(* PLC project abak_app511_10v 0.0.5.project, Abak.IDE Abak.IDE V1.0.0.0 *)
(* stored: creationDateTime 2026-06-29T13:49:17.1967316, modificationDateTime 2026-06-29T10:17:52.4593439 *)

{attribute 'pack_mode' := '1'}
TYPE Coils :
STRUCT
// --- Режимы работы (команды из HMI) ---
xManualMode_Diazo   : BOOL;        // 1. Ручной режим Diazo
xManualMode_Soda    : BOOL;        // 2. Ручной режим Soda
xManualMode_Steam   : BOOL;        // 3. Ручной режим Steam
// --- Управление водой имитатором ---
xWaterValve_AutoMode : BOOL;       // 4. TRUE=Автоматический режим, FALSE=Ручной
xWaterValve_HmiOpen  : BOOL;       // 5. Открытие по кнопке из HMI (в ручном режиме)
xWaterValve_AutoReq  : BOOL;       // 6. Запрос на открытие от автоматики
// --- Сигналы запуска ---
xWaterStart          : BOOL;       // 7. Запуск дозы воды из HMI
xStartHeating_511    : BOOL;       // 8. Запуск прогрева
// --- Сигналы и статусы стадии промывки (Cascade Drain) ---
xStartCoupling_511   : BOOL;       // 9. Запуск с HMI: признак запуска стадии промывки
xCouplingActive_511  : BOOL;       // 10. Статус для HMI: признак "работа идет"
xCouplingDone_511    : BOOL;       // 11. Статус для HMI: признак "успешно готово"
// --- Режим удержания температуры ---
xKeepTempHeating_511 : BOOL;       // 12. TRUE = удержание температуры после нагрева, FALSE = разовый нагрев
// --- Служебные ---
PLC_READ             : BOOL := TRUE; // 13. Флаг чтения PLC
END_STRUCT
END_TYPE

{attribute 'pack_mode' := '4'}
TYPE HoldingRegs : 
STRUCT
// =============================================================
// Модули M7–M9 (MDS AO-2UI) - Управление клапанами (Выходы 4-20мА)
// =============================================================

// --- Управление запорно-регулирующими клапанами (задание 0..100%) ---
AO1_CmdValveDiazo   : REAL;    // 101. Управление клапаном диазосоединения
AO2_CmdValveSoda    : REAL;    // 103. Управление клапаном едкого натра 14%
AO3_CmdValveSteam   : REAL;    // 105. Управление клапаном пара 6 ати

// --- Уставки с панели (ручной режим) ---
rValveManSet_Diazo  : REAL := 0.0;    // 107. Уставка с панели: Диазо
rValveManSet_Soda   : REAL := 0.0;    // 109. Уставка с панели: Сода
rValveManSet_Steam  : REAL := 0.0;    // 111. Уставка с панели: Пар

// --- Переменные для автоматического управления (выходы ПИД-регуляторов) ---
rAutoSet_Diazo      : REAL;           // 113. Выход ПИД расхода диазо
rAutoSet_Soda       : REAL;           // 115. Выход ПИД расхода соды
rAutoSet_Steam      : REAL;           // 117. Выход ПИД расхода пара

// --- Технологические уставки ---
rWaterDose          : REAL := 5.0;    // 119. Заданная доза воды, м³ (5 кубов)
rSetTempApp511      : REAL := 86.0;   // 121. Уставка температуры
rSetFlowDiazo_511   : REAL;           // 123. Уставка мгновенного расхода диазосоединения (до 19 м³/ч)
rSetPh_511          : REAL;           // 125. Целевая уставка pH (9.5..12 ед.)

// --- Настройки алгоритма опустошения емкости (для наладчика) ---
rZeroFlowThreshold_511 : REAL := 0.2; // 127. Порог падения расхода диазо (м³/ч), ниже которого считаем, что емкость пуста
uiEmptyDelaySec_511    : UINT := 20;  // 129. Задержка фиксации пустого трубопровода (сек)

// --- Настройки ПИД-регуляторов (для наладки контуров с HMI) ---
rKp_Diazo_511        : REAL := 1.0;   // 131. Пропорциональный коэффициент контура расхода диазосоединения
rTn_Diazo_511        : REAL := 5.0;   // 133. Время интегрирования контура расхода диазосоединения (сек)
rKp_pH_511           : REAL := 2.0;   // 135. Пропорциональный коэффициент контура pH
rTn_pH_511           : REAL := 10.0;  // 137. Время интегрирования контура pH (сек)
rKp_Steam_511        : REAL := 2.0;   // 139. Пропорциональный коэффициент контура пара (нагрева)
rTn_Steam_511        : REAL := 15.0;  // 141. Время интегрирования контура пара (сек)
rTv_Steam_511        : REAL := 0.0;   // 143. Время дифференцирования контура пара (сек)

END_STRUCT
END_TYPE

{attribute 'pack_mode' := '4'}
TYPE InputRegs : 
STRUCT
	COILS : DINT := 0;
	INPUTS: DINT := 0;
	HOLDINGS: DINT := 0;
	INPUTREGS: DINT := 0;
	
  // МОДУЛЬ АНАЛОГОВЫХ ВХОДОВ (AI)
  	{region M1_K3_AI_10_08_00 }
    // =========================================================================
    // Первые 3 канала: Сигнализация положений (% открытия) клапанов [1, 2]
    (* adr 9 *)  rPosValveDiazo  : REAL; // Канал 1: Обратная связь клапана диазосоединения
    (* adr 11 *) rPosValveSoda   : REAL; // Канал 2: Обратная связь клапана едкого натра 14%
    (* adr 13 *) rPosValveSteam  : REAL; // Канал 3: Обратная связь клапана пара
    
    // Канал 4: рН-метр
    (* adr 15 *) rPhApp511       : REAL; // Канал 4: Показания pH-метра аппарата 511 (диапазон 9,5..12 ед.)
			{endregion}
				 
				 
				 
	{region M5_MDS_3RTD_1 }
	(* adr 17 *) rTempApp511     : REAL; // Температура в аппарате 511 (до 100 С°)
				
   	{endregion}
		 
	{region tenzo tv006c }
	(* adr 19 *) WE_1            : REAL;
	(* adr 21 *) WE_2            : REAL;
		 
   	{endregion}
		 		 
	{region tenzo ELMER }

	(* adr 23 *) IR_FlowSoda   : REAL; // Текущий расход щелочи , л/мин (или м3/ч)
	(* adr 25 *) IR_TotalSoda   : REAL; // Накопленный объем щелочи, л (или м3)
	(* adr 27 *) IR_FlowWater     : REAL; // Текущий расход воды, л/мин (или м3/ч)
	(* adr 29 *) IR_TotalWater   : REAL; // Накопленный объем воды, л (или м3)
		 
    // Выходные сигналы загрузки воды
	(* adr  31*)   rWaterLoaded   : REAL;    // Сколько воды загружено, м³
	(* adr 32*)    rWaterStatus   : REAL;    // Статус загрузки воды: 0=IDLE 1=RUNNING 2=DONE 3=ABORTED
		 
	(* adr  33*)  IR_FlowDiazo   : REAL; // Текущий мгновенный расход диазосоединения (м3/ч) [3]
	(* adr  35*)  IR_TotalDiazo   : REAL; // Текущий расход диазосоединения, л/мин (или м3/ч)
		 
	(* adr  37*)  rDizoStatus   : REAL; // Текущий расход диазосоединения, л/мин (или м3/ч)

	(* adr  39*) rDiazoLoaded   : REAL; // Текущий расход диазосоединения, л/мин (или м3/ч)
rTimeLeft_511:REAL ;///Оставшиеся секунды при падении расхода
	 rStateCode_511:REAL;//
		  
   	{endregion}
		 
END_STRUCT
END_TYPE

{attribute 'pack_mode' := '1'}
TYPE Inputs : 
STRUCT	
			// =============================================================
			// Модуль M11 (MDS DIO-16BD) - Статусы насосов (Дискретные входы)
			// =============================================================
			{region M11 - MDS DIO-16BD (Статусы насосов)}

		
				     
    // Выходная переменная на физическое реле/соленоид
    xWaterValve_Out     : BOOL;  // 1 канал ФЕ
	xWaterValve_SQH :BOOL;
	xWaterValve_SQL   :BOOL;
			{endregion}
END_STRUCT
END_TYPE

TYPE E_InfluxType :
(
    REAL_TYPE,
    INT_TYPE,
    BOOL_TYPE
);
END_TYPE

TYPE E_AO_State :
(
    INIT    := 0,       // Проверка готовности указателей
    IDLE    := 1,       // Ожидание и циклическое обновление
    ERROR   := 99       // Ошибка адресации или данных
) INT;
END_TYPE

{attribute 'qualified_only'}
{attribute 'strict'}
TYPE E_ValveMode :
(
    INIT := 0,
    AUTO := 1,
    MANUAL := 2,
    ERROR := 99
) INT; // Указываем базовый тип для совместимости
END_TYPE

TYPE E_PumpState :
(
    INIT,           // Инициализация и проверка ресурсов
    IDLE,           // Ожидание команды
    START_PULSE,    // Формирование импульса на ПУСК
    STOP_PULSE,     // Формирование импульса на СТОП
    BLIND_WINDOW,   // Окно игнорирования изменений (x2 времени импульса)
    ERROR           // Состояние критической ошибки
);
END_TYPE

TYPE E_TempSourceSelect_for_cube :
(
   AI_T2_Temp_Cube := 0,  // Температура в кубе
    AI_T3_Temp_Packing := 1,  // T3: Температура в нижней части насадки
    AI_T4_Temp_BotCol := 2   // [Канал 1] T4: Температура низа колонны
) INT;
END_TYPE

{attribute 'qualified_only'}
{attribute 'strict'}
TYPE E_ValveState :
(
    INIT    := 0,   // Инициализация указателей
    IDLE    := 1,   // Ожидание выбора режима
    AUTO    := 2,   // Автоматическое управление
    MANUAL  := 3,   // Ручное управление (HMI)
    FAULT   := 99   // Состояние ошибки (например, Null Pointer)
);
END_TYPE

TYPE E_InfluxType_1 :
(
    REAL_TYPE,
    INT_TYPE,
    BOOL_TYPE
);
END_TYPE

// шаг состояния клиента
{attribute 'strict'}
TYPE CLIENT_STATE :
(
	CREATE	:=	 0,
	WAITING	:=	10,
	SEND	:=	20,
	RECEIVE :=  30
);
END_TYPE

TYPE E_REM_State :
(
    INIT,              (* Начальная инициализация и сброс регистров при запуске *)
    OPERATING,         (* Нормальный циклический режим обработки физических данных *)
    RESET_LOGIC,       (* Шаг удержания команды сброса сумматора *)
    ERROR_COMM         (* Состояние аварии связи при отказе Modbus-канала *)
)  := INIT;            (* По умолчанию автомат всегда стартует с шага INIT *)
END_TYPE

TYPE U_WordToReal : UNION
  dwValue : DWORD;  (* Используется для битовых операций *)
  rValue : REAL;  (* Используется для получения результата *)
END_UNION;
END_TYPE

PROGRAM PLC_PRG // Antigravity Sync Test
VAR
    fbElemerREM         : fbElemerREM;
    
    (* Переменные из вкладки Modbus Generic Serial Slave I/O Mapping *)
    Hmi_Flow_Regs    AT %IW67  : ARRAY[0..1] OF WORD; (* Канал 0 (Мгновенный расход) *)
    Hmi_Volume_Regs  AT %IW63  : ARRAY[0..3] OF WORD; (* Канал 1 (Накопленный объем) *)
    xModbusCommError    : BOOL;                 (* Системный флаг ошибки связи с прибором *)
    xHmiResetCmd        : BOOL;                 (* Сигнал сброса сумматора с HMI-панели *)
    
    (* Выходные очищенные технологические переменные *)
    rCurrentFlowRate    : REAL;                 (* Мгновенный расход в систему, куб.м/ч *)
    lrAccumulatedVol    : LREAL;                (* Точный накопленный объем, куб.м *)
    sOperatorMessage    : STRING(255);          (* Сообщение для текстовой строки на панели *)

    fbWater             : FB_WaterLoading;      (* Наш исправленный ФБ дозирования *)
    
    // ============================================================
    // ПЕРЕМЕННЫЕ ДЛЯ ТЕСТИРОВАНИЯ И СИМУЛЯЦИИ СУММАТОРА
    // ============================================================
    xSimEnable          : BOOL := FALSE;        (* Включить режим симуляции (True = подмена датчиков) *)
    rSimFlowSpeed       : REAL := 20.0;         (* Скорость потока при открытом клапане, куб.м/ч *)
    rSimTotalStorage    : REAL := 125.45;       (* Внутренний виртуальный накопительный счетчик куб.м *)
    
    fbSimClock          : TON;                  (* Генератор тактов времени для подсчета объема *)
    rDeltaVolume        : REAL;                 (* Математический шаг приращения за 1 такт *)
    // ============================================================
END_VAR

                  // ================================================================
// 1. ЧТЕНИЕ РЕАЛЬНЫХ ДАННЫХ ИЗ ПОЛЕВЫХ ПРИБОРОВ
// ================================================================
gvl.gInputRegs.IR_TotalSoda := F_ElemerREM_Volume(pBuf := ADR(%IW65));
gvl.gInputRegs.IR_FlowSoda  := F_ElemerREM_Flow(pBuf := ADR(%IW69));
gvl.gInputRegs.rTempApp511  := F_GetReal_BADC(pBuf := ADR(%IW57));


// ================================================================
// 2. ДИНАМИЧЕСКИЙ СИМУЛЯТОР РАСХОДОМЕРА ВОДЫ
// ================================================================
// Тактовый генератор: срабатывает каждые 100 мс (0.1 секунды) для плавности хода счета
fbSimClock(IN := xSimEnable AND NOT fbSimClock.Q, PT := T#100ms);

IF xSimEnable THEN
    // ЕСЛИ СИМУЛЯЦИЯ ВКЛЮЧЕНА:
    
    // Имитируем поведение потока в зависимости от команды на клапан
    IF gvl.gCoils.xWaterValve_AutoReq THEN
        // Клапан открыт автоматикой -> задаем симуляционный расход
        gvl.gInputRegs.IR_FlowWater := rSimFlowSpeed; 
        
        // Расчет приращения сумматора за 100мс: (куб.м/ч * 0.1с) / 3600с
        IF fbSimClock.Q THEN
            rDeltaVolume := (rSimFlowSpeed * 0.1) / 3600.0;
            rSimTotalStorage := rSimTotalStorage + rDeltaVolume;
        END_IF;
    ELSE
        // Клапан закрыт -> поток прекращается
        gvl.gInputRegs.IR_FlowWater := 0.0;
    END_IF;

    // ПОДМЕНЯЕМ значение сумматора результатом симуляции для ФБ дозирования
    gvl.gInputRegs.IR_TotalWater := rSimTotalStorage;

ELSE
    // ЕСЛИ СИМУЛЯЦИЯ ВЫКЛЮЧЕНА (РАБОЧИЙ РЕЖИМ):
    
    // Читаем физический прибор с адреса %IW71 и %IW75
    gvl.gInputRegs.IR_TotalWater := F_ElemerREM_Volume(pBuf := ADR(%IW71));
    gvl.gInputRegs.IR_FlowWater  := F_ElemerREM_Flow(pBuf := ADR(%IW75));
    
    // Мягко синхронизируем симулятор, чтобы при включении тумблера счет не прыгал назад/вперед
    rSimTotalStorage := gvl.gInputRegs.IR_TotalWater;
END_IF;


// ================================================================
// 3. ВЫЗОВ И ПРОВЕРКА ФУНКЦИОНАЛЬНОГО БЛОКА ЗАГРУЗКИ ВОДЫ
// ================================================================
fbWater(
    rTotalVolume := gvl.gInputRegs.IR_TotalWater,        // Сюда идет либо физический объем, либо симуляция
    rDose        := gvl.gHoldingRegs.rWaterDose,         // Заданная уставка дозы (куб.м)
    rDeadband    := 0.05,                                // Упреждение закрытия (0.05 куб.м)
    xStart       := gvl.gCoils.xWaterStart,              // Команда Старт/Стоп
    xMode        := gvl.gCoils.xWaterValve_AutoMode,     // Флаг режима АВТО клапана
    xAutoControl := gvl.gCoils.xWaterValve_AutoReq       // Управление клапаном (выход на открытие)
);

    gvl.gInputRegs.rWaterLoaded:=fbWater.rLoaded;
    gvl.gInputRegs.rWaterStatus:=fbWater.rStatus;
                
END_PROGRAM

FUNCTION AIToFloat : REAL
VAR_INPUT
	In:UINT;
	Lo,Hi:REAL;
END_VAR
VAR
END_VAR

                  AIToFloat:=(UINT_TO_REAL(In)-10000.0)/40000.0*Hi+Lo;
//AIToFloat:=(UINT_TO_REAL(In)-0.0)/50000.0*Hi+Lo;
                
END_FUNCTION

PROGRAM ASK_prg
VAR
Exatract:	FB_ModbusToFloatArray;
pt : POINTER TO  ARRAY [0..5] OF WORD  ;

//M1_K3_AI_10_08_00 AT %IW58: ARRAY [0..7] OF WORD ; 

buff_abak: ARRAY [0..219] OF WORD ; 
buff_MDS: ARRAY [0..219] OF WORD ; 
buffR_1: ARRAY [0..119] OF REAL ; 
start_ad_mds3rtd:INT:=0;
swap_mds3rtd:INT:=6;
start_ad_mds_8UId:INT:=18;
swap_mds_8UI:INT:=16;

AI: FB_AI;


  
	Info : __SYSTEM.VAR_INFO;

    pAddress : POINTER TO BYTE;
	adress:UDINT;
END_VAR

                  //берем  с модуля  M1_K3_AI_10_08_00 значения  и  копируем в промежуточный буфер   
SysMemCpy(ADR(buff_abak), ADR( %IW0), 8 * SIZEOF(WORD));

//берем  с модуля  MDS_3RTD_1  значения  и  копируем в промежуточный буфер   
SysMemCpy(ADR(buff_MDS), ADR( %IW57), 6 * SIZEOF(WORD));


//берем  с  терминала  tv 006
SysMemCpy(ADR(buff_MDS[swap_mds3rtd]), ADR( %IW53), 2* SIZEOF(WORD));

//берем  с  терминала  tv 006
SysMemCpy(ADR(buff_MDS[swap_mds3rtd+2]), ADR( %IW55), 2* SIZEOF(WORD));

Exatract(aDataIn:=buff_MDS,aDataOut=>buffR_1,IQty:=65,iMode:=1);


// 3. Маппинг (Присвоение значений переменным структуры)
// -------------------------------------------------------------

// === Модуль M1 () ===
GVL.gInputRegs. rPosValveDiazo  := AIToFloat(buff_abak[0],0,100); // 
GVL.gInputRegs.rPosValveSoda  := AIToFloat(buff_abak[1],0,100); // 
GVL.gInputRegs.rPosValveSteam  := AIToFloat(buff_abak[2],0,100); // 
GVL.gInputRegs.rPhApp511  := AIToFloat(buff_abak[4],0,14); // 


// === Модуль M5 () ===

GVL.gInputRegs.rTempApp511  :=buffR_1[0];// TT 511
//GVL.gInputRegs.rTempApp511  :=FC_ModbusToRealSwapped(wWord1 := buff_MDS[0], wWord2 := buff_MDS[1]);
// === Модуль M2 () ===
GVL.rCmdValveDiazo := FloatToAI(gvl.gHoldingRegs.AO1_CmdValveDiazo);

GVL.rCmdValveSoda := FloatToAI(gvl.gHoldingRegs.AO2_CmdValveSoda);

GVL.rCmdValveSteam := FloatToAI(gvl.gHoldingRegs.AO3_CmdValveSteam);


// === Модуль M5 (Индексы 0..2) ===
//GVL.gInputRegs.rTempApp511   := buffR_1[0]; // TT 511


//// === весы  tenzo  M1 ===

	//AI(F_WORD_IN:= gvl.WE_1_f, S_WORD_IN:= gvl.WE_1_s, RANGE_CONV:=FALSE, VAL_OUT=> GVL.gInputRegs.WE_1);
GVL.gInputRegs.WE_1:=buffR_1[3];
GVL.gInputRegs.WE_2:=buffR_1[4];
//// === весы  tenzo  M2 ===
//AI(F_WORD_IN:= gvl.WE_2_f, S_WORD_IN:= gvl.WE_2_s, RANGE_CONV:=TRUE, VAL_OUT=> GVL.gInputRegs.WE_2);
                
END_PROGRAM

FUNCTION_BLOCK FB_ModbusToFloatArray
VAR_INPUT
    aDataIn : ARRAY [0..219] OF WORD; // Входной массив (до 120 регистров)
    iQty    : INT := 1;               // Количество FLOAT переменных для обработки (макс 60)
    iMode   : INT := 1;               // Режим: 0=1234, 1=3412 (частый), 2=2143, 3=4321
END_VAR
VAR_OUTPUT
    aDataOut : ARRAY [0..119] OF REAL; // Выходной массив
    xError   : BOOL;                  // Флаг ошибки (если iQty > 60)
END_VAR
VAR
    i : INT;
    uConverter : U_WordToReal;
    wLow : WORD;
    wHigh : WORD;
    wTemp1 : WORD;
    wTemp2 : WORD;
END_VAR

                  
// Сброс ошибки
xError := FALSE;

// Защита от выхода за пределы массива
IF iQty < 1 OR iQty > 120 THEN
    xError := TRUE;
    RETURN;
END_IF

// Основной цикл
FOR i := 0 TO (iQty - 1) DO
    
    // Получаем пару регистров из массива
    // i*2 - это начало пары (0, 2, 4...)
    wTemp1 := aDataIn[i * 2];     // Первый регистр пары
    wTemp2 := aDataIn[(i * 2) + 1]; // Второй регистр пары

    CASE iMode OF
        // ---------------------------------------------------------
        // Mode 0: 1234 (Big Endian) 
        // Порядок: [HighWord] [LowWord]
        // ---------------------------------------------------------
        0: 
            wHigh := wTemp1;
            wLow  := wTemp2;
            
        // ---------------------------------------------------------
        // Mode 1: 3412 (Middle Little / Word Swap) -> САМЫЙ ЧАСТЫЙ для Modbus
        // Порядок: [LowWord] [HighWord]
        // Регистры меняются местами, байты внутри - нет.
        // ---------------------------------------------------------
        1: 
            wHigh := wTemp2;
            wLow  := wTemp1;

        // ---------------------------------------------------------
        // Mode 2: 2143 (Middle Big / Byte Swap)
        // Порядок: [HighWord swapped] [LowWord swapped]
        // Байты меняются местами внутри каждого слова.
        // ---------------------------------------------------------
        2:
            wHigh := ROL(wTemp1, 8); // Меняем байты местами
            wLow  := ROL(wTemp2, 8);
            
        // ---------------------------------------------------------
        // Mode 3: 4321 (Little Endian)
        // Порядок: [LowWord swapped] [HighWord swapped]
        // Полный разворот: меняются и слова, и байты.
        // ---------------------------------------------------------
        3:
            wHigh := ROL(wTemp2, 8);
            wLow  := ROL(wTemp1, 8);
            
        ELSE
            // По умолчанию используем 3412 (как самый популярный)
            wHigh := wTemp2;
            wLow  := wTemp1;
    END_CASE

    // Сборка DWORD из двух слов
    // Сдвигаем старшее слово на 16 бит влево и добавляем младшее
    uConverter.dwValue := SHL(WORD_TO_DWORD(wHigh), 16) OR WORD_TO_DWORD(wLow);
    
    // Запись результата в выходной массив
    aDataOut[i] := uConverter.rValue;
    
END_FOR
                
END_FUNCTION_BLOCK

FUNCTION_BLOCK Check_Block
VAR_INPUT
	State_Mixer : BOOL;
	Weight : REAL;
END_VAR
VAR_OUTPUT
	State_Block : BOOL;
	State_Block_P102 : BOOL; 
END_VAR
VAR
END_VAR

                  IF NOT State_Mixer THEN
	State_Block := TRUE;
ELSE
	State_Block := FALSE;
END_IF;
IF Weight > 3000 THEN
	State_Block_P102 := TRUE;
ELSE 
	State_Block_P102 := FALSE;
END_IF;
                
END_FUNCTION_BLOCK

FUNCTION FloatToAI : UINT
VAR_INPUT
	In:REAL;
	
END_VAR
VAR
END_VAR

                  FloatToAI:=REAL_TO_UINT(In/100.0*40000.0+10000.0);
                
END_FUNCTION

(*
* @fb: PRG_ModbusSlave_Sync
* @desc: Исправленная синхронизация через прямые указатели (устранение C0047/C0077)
*)
PROGRAM PRG_ModbusSlave_Sync
VAR
    fbSlv               : abakplcutils.MDB;
    sStatus             : STRING(255);
    
    // Вспомогательные буферы
    wMbHolding          : ARRAY[0..500] OF WORD; 
    wOldMbHolding       : ARRAY[0..500] OF WORD; 
    
    // Указатели для работы со структурами GVL как с массивами
    pCurrWord           : POINTER TO WORD;
    pOldWord            : POINTER TO WORD;
    
    wIndex              : WORD;
    uiHoldRegsCnt       : WORD;
    uiInRegsCnt         : WORD;
    xFirstLoop          : BOOL := TRUE;
	
    C_INPUT_REG_START   : WORD := 1;
    C_HOLD_REG_START    : WORD := 1000;
END_VAR

                  // 1. Инициализация и расчет длин (через SIZEOF, чтобы не зависеть от типов)
IF xFirstLoop THEN
    uiInRegsCnt   := ANY_TO_WORD(SIZEOF(GVL.gInputRegs) / 2);
    uiHoldRegsCnt := ANY_TO_WORD(SIZEOF(GVL.gHoldingRegs) / 2);
    
    // Предзаполнение Modbus и локального зеркала (используем SysMem для скорости)
    fbSlv.SetWordRegs(reg := C_HOLD_REG_START, pBuf := ADR(GVL.gHoldingRegs), cnt := uiHoldRegsCnt);
    SysMem.SysMemCpy(pDest := ADR(wOldMbHolding), pSrc := ADR(GVL.gHoldingRegs), udiCount := uiHoldRegsCnt * 2);
    
    xFirstLoop := FALSE;
    RETURN;
END_IF

// --- ШАГ 1: Input Registers (Запись всей структуры целиком через указатель) ---
sStatus := 'Обновление Input Registers';
fbSlv.SetWordRegs(reg := C_INPUT_REG_START, pBuf := ADR(GVL.gInputRegs), cnt := uiInRegsCnt);

// --- ШАГ 2: Holding Registers (Синхронизация через пошаговый доступ к памяти) ---
sStatus := 'Синхронизация Holding...';
fbSlv.GetWordRegs(reg := C_HOLD_REG_START, pBuf := ADR(wMbHolding), cnt := uiHoldRegsCnt);

FOR wIndex := 0 TO (uiHoldRegsCnt - 1) DO
    // Получаем адреса текущего слова в GVL и в нашем зеркале Old
    pCurrWord := ADR(GVL.gHoldingRegs) + (wIndex * 2); // Смещение в байтах (WORD = 2 байта)
    pOldWord  := ADR(wOldMbHolding) + (wIndex * 2);

    // Сценарий А: Изменение в ПЛК
    IF pCurrWord^ <> pOldWord^ THEN
        fbSlv.SetWord(reg := C_HOLD_REG_START + wIndex, val := pCurrWord^);
        pOldWord^ := pCurrWord^; // Обновляем зеркало
        
    // Сценарий Б: Изменение в Modbus (от SCADA)
    ELSIF wMbHolding[wIndex] <> pOldWord^ THEN
        pCurrWord^ := wMbHolding[wIndex]; // Пишем напрямую в структуру GVL
        pOldWord^  := wMbHolding[wIndex]; // Обновляем зеркало
    END_IF
END_FOR

// Синхронизация с энергонезависимой памятью
PVL.rHoldingRegs := GVL.gHoldingRegs;
                
END_PROGRAM

PROGRAM PLC_PRG_MBS_TCP_SLAVE
VAR
	bFirstLoop	: BOOL := FALSE;
	fbSlv		: AbakPLCUtils.MDB;	
	
	pInputRegs			:	POINTER TO WORD;
	wInputRegsLength	:	WORD 	:= SIZEOF(GVL.gInputRegs)/2;
	
	pHoldingRegs			:	POINTER TO WORD;
	wHoldingRegsLength	:	WORD 	:= SIZEOF(GVL.gHoldingRegs)/2;
	
	pInputs			:	POINTER TO BOOL;
	wInputsLength	:	WORD 	:= SIZEOF(GVL.gInputs);
	
	pCoils			:	POINTER TO BOOL;
	wCoilsLength	:	WORD 	:= SIZEOF(GVL.gCoils);
	
	wIndex		:	WORD := 0; 
	
	pMbHolding			:	POINTER TO WORD;
	pOldMbHoldingRegs			:	POINTER TO WORD;
	pOldHoldingRegs			:	POINTER TO WORD;
	
	wMbHolding	:   ARRAY[0..1] OF WORD;
	wOldMbHoldingRegs	:   ARRAY[0..( SIZEOF(GVL.gHoldingRegs)/2-1)] OF WORD;
	wOldHoldingRegs	:   ARRAY[0..(SIZEOF(GVL.gHoldingRegs)/2-1)] OF WORD;
	
	pMbCoil		:	POINTER TO BOOL;
	pOldMbCoils			:	POINTER TO BOOL;
	pOldCoils			:	POINTER TO BOOL;
	
	bMbCoil	:   ARRAY[0..0] OF BOOL;
	bOldMbCoils	:   ARRAY[0..(SIZEOF(GVL.gCoils) -1)] OF BOOL;
	bOldCoils	:   ARRAY[0..(SIZEOF(GVL.gCoils) -1)] OF BOOL;
	
	bIsGetMb: BYTE := 0;
	
	    wInputRegsOffset    : WORD := 0;  // InputRegs начинаются с адреса 1000
    wInputsOffset       : WORD := 499;   // Inputs начинаются с адреса  
    wHoldingRegsOffset  : WORD := 100;     // HoldingRegs - без смещения (или задай своё)
    wCoilsOffset        : WORD := 0;     // Coi
END_VAR

                  IF NOT bFirstLoop THEN
	fbSlv.IsVirtualModbus := 0;
	
	GVL.gInputRegs.INPUTREGS := SIZEOF(GVL.gInputRegs)/2;
	GVL.gInputRegs.HOLDINGS := SIZEOF(GVL.gHoldingRegs)/2;
	GVL.gInputRegs.INPUTS := SIZEOF(GVL.gInputs);
	GVL.gInputRegs.COILS := SIZEOF(GVL.gCoils);
	
	MBS_HoldingRegs_Change();
	MBS_Coils_Change();
	
	GVL.gHoldingRegs :=PVL.rHoldingRegs;
	bFirstLoop := TRUE;
ELSE
	MBS_HoldingRegs_Change();
	MBS_Coils_Change();

	MBS_InputRegs_WRITE();
	MBS_Inputs_WRITE();
	PVL.rHoldingRegs :=GVL.gHoldingRegs;
END_IF
                

ACTION MBS_InputRegs_WRITE:
                      wIndex := 0;
pInputRegs := ADR(GVL.gInputRegs);

//WHILE wIndex < wInputRegsLength DO
	fbSlv.SetWordRegs (wInputRegsOffset +wIndex + 1 , pInputRegs, wInputRegsLength);	

	// INC
	//wIndex := wIndex + 1;
//	pInputRegs := pInputRegs + SIZEOF(WORD);
//END_WHILE;

                    
END_ACTION

ACTION MBS_HoldingRegs_Change:
                      wIndex :=0;
pHoldingRegs:= ADR(GVL.gHoldingRegs);
pMbHolding := ADR(wMbHolding);
pOldMbHoldingRegs:= ADR(wOldMbHoldingRegs);
pOldHoldingRegs	:= ADR(wOldHoldingRegs);

WHILE wIndex < wHoldingRegsLength DO
	
	wMbHolding[0]:= 0;
	wMbHolding[1]:= 0;	
	IF NOT bFirstLoop THEN
		fbSlv.SetWordRegs(wHoldingRegsOffset + wIndex + 1 , pMbHolding, 2);	
		MEMUtils.MemCpy(pbyDest := pOldMbHoldingRegs, pbySrc := pMbHolding, 4);
		MEMUtils.MemCpy(pbyDest := pOldHoldingRegs, pbySrc := pMbHolding, 4);	
	ELSE
		bIsGetMb := fbSlv.GetWordRegs(wHoldingRegsOffset  + wIndex + 1,  pMbHolding, 2);
	
		IF (NOT MEMUtils.MemCmp(pOldHoldingRegs, pHoldingRegs,4)) THEN
			
			MEMUtils.MemCpy(pbyDest := pMbHolding, pbySrc := pHoldingRegs, 4);
			fbSlv.SetWordRegs(wHoldingRegsOffset + wIndex + 1 , pMbHolding, 2);	
			
		ELSIF (NOT MEMUtils.MemCmp(pOldMbHoldingRegs, pMbHolding,4)) THEN
			
			MEMUtils.MemCpy(pbyDest := pHoldingRegs, pbySrc := pMbHolding, 4);
		END_IF
		
		MEMUtils.MemCpy(pbyDest := pOldMbHoldingRegs, pbySrc := pMbHolding, 4);
		MEMUtils.MemCpy(pbyDest := pOldHoldingRegs, pbySrc := pHoldingRegs, 4);
	END_IF
	// INC		
 	wIndex := wIndex + 2;
	
	pOldMbHoldingRegs:= pOldMbHoldingRegs + 4;
	pOldHoldingRegs:= pOldHoldingRegs + 4;
    pHoldingRegs := pHoldingRegs + 4;
END_WHILE;
                    
END_ACTION

ACTION MBS_Inputs_WRITE:
                      wIndex := 0;
pInputs := ADR(GVL.gInputs);

WHILE wIndex < wInputsLength DO
	bMbCoil[0] := pInputs^;
	fbSlv.SetCoil(wInputsOffset + wIndex + 1 , pInputs^);	

	// INC
	wIndex := wIndex + 1;
	pInputs := pInputs + SIZEOF(BOOL);
END_WHILE;

                    
END_ACTION

ACTION MBS_Coils_Change:
                      wIndex := 0;
pCoils := ADR(GVL.gCoils);

pMbCoil := ADR(bMbCoil);
pOldMbCoils:= ADR(bOldMbCoils);
pOldCoils	:= ADR(bOldCoils);

WHILE wIndex < wCoilsLength DO
	IF NOT bFirstLoop THEN
		pMbCoil^:=FALSE;
		fbSlv.SetCoil(wCoilsOffset  + wIndex + 1 , pMbCoil^);
		MEMUtils.MemCpy(pbyDest := pOldMBCoils, pbySrc := pMbCoil, 1);
		MEMUtils.MemCpy(pbyDest := pOldCoils, pbySrc := pMbCoil, 1);	
	ELSE
	
		pMbCoil^ := fbSlv.GetCoil(wCoilsOffset  + wIndex + 1);
	
		IF (NOT MEMUtils.MemCmp(pOldCoils, pCoils, 1)) THEN
			
			MEMUtils.MemCpy(pbyDest := pMbCoil, pbySrc := pCoils, 1);
			fbSlv.SetCoil(wCoilsOffset  + wIndex + 1 , pMbCoil^);	
			
		ELSIF (NOT MEMUtils.MemCmp(pOldMbCoils, pMbCoil, 1)) THEN
			
			MEMUtils.MemCpy(pbyDest := pCoils, pbySrc := pMbCoil, 1);
		END_IF
		
		MEMUtils.MemCpy(pbyDest := pOldMBCoils, pbySrc := pMbCoil, 1);
		MEMUtils.MemCpy(pbyDest := pOldCoils, pbySrc := pCoils, 1);
	END_IF
	// INC		
 	wIndex := wIndex + 1;
	
	pOldMbCoils:= pOldCoils + 1;
	pOldCoils:= pOldCoils + 1;
    pCoils := pCoils + 1;
END_WHILE;
                    
END_ACTION
END_PROGRAM

(*
    Название: FB_ValveLogic
    Автор: Gemini Industrial AI
    Версия: 1.1.0
    Описание: Управление клапаном с прямой записью REAL значения через указатель.
*)
FUNCTION_BLOCK FB_ValveLogic
VAR_INPUT
    xModeManual     : BOOL;             // Переключатель: TRUE - Ручной, FALSE - Авто
    xEnableLog      : BOOL := TRUE;     // Разрешить текстовое логирование
    rMinLimit       : REAL := 0.0;      // Нижний предел уставки
    rMaxLimit       : REAL := 100.0;    // Верхний предел уставки (например, 100%)
END_VAR

VAR_OUTPUT
    sStatus         : STRING(80);       // Диагностика на русском языке
    rActualSetpoint : REAL;             // Текущая выбранная уставка
    xError          : BOOL;             // Флаг ошибки указателей
END_VAR

VAR
    (* Указатели *)
    pSetMan         : POINTER TO REAL;  // Ссылка на ручную переменную (HMI)
    pSetAuto        : POINTER TO REAL;  // Ссылка на авто переменную (PID)
    pOutReal        : POINTER TO REAL;  // Ссылка на выходную переменную REAL
    
END_VAR

                  // 1. Проверка инициализации основного выходного указателя
IF pOutReal = 0 THEN
    xError := TRUE;
    sStatus := 'ОШИБКА: Целевой адрес OutReal не назначен!';
    RETURN; // Прекращаем выполнение, чтобы не вызвать исключение
END_IF

// 2. Выбор источника данных в зависимости от режима
IF xModeManual THEN
    // Режим РУЧНОЙ
    IF pSetMan <> 0 THEN
        rActualSetpoint := pSetMan^;
        xError := FALSE;
        IF xEnableLog THEN sStatus := 'Режим: РУЧНОЙ. Уставка с HMI.'; END_IF
    ELSE
        xError := TRUE;
        sStatus := 'Ошибка: Пустой указатель на ручную уставку!';
    END_IF
ELSE
    // Режим АВТО
    IF pSetAuto <> 0 THEN
        rActualSetpoint := pSetAuto^;
        xError := FALSE;
        IF xEnableLog THEN sStatus := 'Режим: АВТО. Управление от ПЛК.'; END_IF
    ELSE
        xError := TRUE;
        sStatus := 'Ошибка: Пустой указатель на авто-уставку!';
    END_IF
END_IF

// 3. Обработка ТАУ (ограничение диапазона)
rActualSetpoint := LIMIT(rMinLimit, rActualSetpoint, rMaxLimit);

// 4. Прямая запись в память по адресу, если нет ошибок
IF NOT xError THEN
    pOutReal^ := rActualSetpoint;
END_IF
                

METHOD PUBLIC Init : BOOL
VAR_INPUT
    pManualVar       : POINTER TO REAL; // Адрес Holding Register (Ручной режим с HMI)
    pAutoVar         : POINTER TO REAL; // Адрес уставки из логики/ПИД (Авто режим)
    pOutputVar       : POINTER TO REAL; // Адрес целевой переменной (куда пишем итог)
END_VAR
                        

pSetMan  := pManualVar;
pSetAuto := pAutoVar;
pOutReal := pOutputVar;

Init := (pSetMan <> 0 AND pSetAuto <> 0 AND pOutReal <> 0);
                      
END_METHOD
END_FUNCTION_BLOCK

FUNCTION FC_Write_AO : BOOL
VAR_INPUT
    VAL_IN  : REAL;    // Входное значение (например, от ПИД 0..1000)

    pOutput : POINTER TO ARRAY[0..1] OF WORD; // Адрес физических регистров модуля
END_VAR
VAR
    TMP     : REAL;
    dwValue : DWORD;
	    X1      : REAL:=0;    // Мин. вход (например, 0)
    X2      : REAL:=100;    // Макс. вход (например, 1000)
    Y1      : REAL:=4;    // Мин. ток (например, 4.0)
    Y2      : REAL:=20;    // Макс. ток (например, 20.0)
END_VAR

                  
// 1. Проверка на нулевой указатель и деление на ноль
IF pOutput = 0 OR (X2 = X1) THEN
    FC_Write_AO := FALSE;
    RETURN;
END_IF;

// 2. Линейное масштабирование (из входного диапазона в 4..20мА)
TMP := (Y2 - Y1) / (X2 - X1) * (VAL_IN - X1) + Y1;

// 3. Преобразование REAL во внутреннее битовое представление DWORD
dwValue := OSCAT_BASIC.REAL_TO_DW(TMP);

// 4. Запись напрямую в память по указателю (разбивка на 2 WORD)
// В ПЛК Абак обычно старшее слово идет первым (зависит от настроек модуля)
pOutput^[0] := OSCAT_BASIC.WORD_OF_DWORD(dwValue, 1); // High Word
pOutput^[1] := OSCAT_BASIC.WORD_OF_DWORD(dwValue, 0); // Low Word

FC_Write_AO := TRUE;
                
END_FUNCTION

FUNCTION FC_Write_AO_CDAB : BOOL
VAR_INPUT
    rValIn   : REAL;    // Входная уставка (0..100)
    pOutput  : POINTER TO ARRAY[0..1] OF WORD; 
    rInMin   : REAL;    
    rInMax   : REAL;    
    rOutMin  : REAL;    
    rOutMax  : REAL;    
END_VAR
VAR
    rScaled  : REAL;
    dwRaw    : DWORD;
	dwCDAB: DWORD;
    pReal    : POINTER TO DWORD;
END_VAR

                  // 1. Линейное масштабирование (Scale)
// Формула: Out = ((In - InMin) * (OutMax - OutMin) / (InMax - InMin)) + OutMin
IF (rInMax <> rInMin) THEN
    rScaled := ((rValIn - rInMin) * (rOutMax - rOutMin) / (rInMax - rInMin)) + rOutMin;
ELSE
    rScaled := rOutMin;
END_IF

// 2. Получаем битовое представление REAL как DWORD
pReal := ADR(rScaled);
dwRaw := pReal^;

// 3. Перепаковка в формат CDAB
// Исходный (ABCD): [Byte3][Byte2][Byte1][Byte0]
// Формат CDAB:     [Byte1][Byte0][Byte3][Byte2]
// То есть меняем местами слова (WORD)

dwCDAB := ROL(dwRaw, 16); // Простейший способ поменять слова местами

// 4. Запись результата по указателю
IF pOutput <> 0 THEN
    pOutput^[1] := DWORD_TO_WORD(dwCDAB AND 16#FFFF);        // Младшее слово CDAB (бывшее старшее AB)
    pOutput^[0] := DWORD_TO_WORD(SHR(dwCDAB, 16));           // Старшее слово CDAB (бывшее младшее CD)
    FC_Write_AO_CDAB := TRUE;
ELSE
    FC_Write_AO_CDAB := FALSE;
END_IF
                
END_FUNCTION

FUNCTION_BLOCK FB_AI
VAR_INPUT
	F_WORD_IN : WORD;
	S_WORD_IN : WORD;
	X1 : REAL:=4;
	Y1 : REAL:=0;
	X2 : REAL:=20;
	Y2 : REAL:=100;
	RANGE_CONV:BOOL:=TRUE;
END_VAR
VAR
	TMP:REAL;
END_VAR
VAR_OUTPUT
	VAL_OUT : REAL;
END_VAR

                  TMP := OSCAT_BASIC.DW_TO_REAL(X:= OSCAT_BASIC.DWORD_OF_WORD(W1:= F_WORD_IN , W0:= S_WORD_IN ));
IF (RANGE_CONV)
THEN
	IF (TMP=9999 OR TMP=-9999 OR TMP=-7777 OR TMP=7777)
	THEN 
		VAL_OUT :=  TMP; 		
	ELSE
		VAL_OUT :=  (Y2 - Y1) / (X2 - X1) * (TMP - X1) + Y1;
	END_IF
	
ELSE
	VAL_OUT :=  TMP; 
END_IF
                
END_FUNCTION_BLOCK

PROGRAM PRG_Valves
VAR

    // Экземпляры логики управления для каждого клапана
    fbValveDiazo : FB_ValveLogic;
    fbValveSoda  : FB_ValveLogic;
    fbValveSteam : FB_ValveLogic;

    // Флаг для однократной инициализации указателей
    xInitDone    : BOOL := FALSE;
    // Экземпляр функционального блока для клапана подачи воды
    fbWaterValve : FB_ValveS_Compact;
    


END_VAR

                  // --- 1. ОДНОКРАТНАЯ ИНИЦИАЛИЗАЦИЯ (Привязка адресов) ---
IF NOT xInitDone THEN
    
    // Привязка для клапана Диазосоединения
    fbValveDiazo.Init(
        pManualVar := ADR(gvl.gHoldingRegs.rValveManSet_Diazo),       // Уставка с HMI
        pAutoVar   := ADR(gvl.gHoldingRegs.rAutoSet_Diazo),     // Уставка от ПИД/Логики
        pOutputVar := ADR(gvl.gHoldingRegs.AO1_CmdValveDiazo)       // Физический выход (M2)
    );

    // Привязка для клапана Едкого натра (Соды)
    fbValveSoda.Init(
        pManualVar := ADR(gvl.gHoldingRegs.rValveManSet_Soda), 
        pAutoVar   := ADR(gvl.gHoldingRegs.rAutoSet_Soda), 
        pOutputVar := ADR(gvl.gHoldingRegs.AO2_CmdValveSoda)        // Физический выход (M2)
    );

    // Привязка для клапана Пара
    fbValveSteam.Init(
        pManualVar := ADR(gvl.gHoldingRegs.rValveManSet_Steam), 
        pAutoVar   := ADR(gvl.gHoldingRegs.rAutoSet_Steam), 
        pOutputVar := ADR(gvl.gHoldingRegs.AO3_CmdValveSteam)       // Физический выход (M2)
    );

    xInitDone := TRUE;
END_IF;

// --- 2. ЦИКЛИЧЕСКИЙ ВЫЗОВ ЛОГИКИ ---

// Управление клапаном Диазосоединения
fbValveDiazo(
    xModeManual :=gvl.gCoils.xManualMode_Diazo,
    rMinLimit   := 0.0,
    rMaxLimit   := 100.0
);

// Управление клапаном Едкого натра
fbValveSoda(
    xModeManual := gvl.gCoils.xManualMode_Soda,
    rMinLimit   := 0.0,
    rMaxLimit   := 100.0
);

// Управление клапаном Пара
fbValveSteam(
    xModeManual := gvl.gCoils.xManualMode_Steam,
    rMinLimit   := 0.0,
    rMaxLimit   := 100.0
);


// Вызов блока управления водяным клапаном
fbWaterValve(
    xMode        := gvl.gCoils.xWaterValve_AutoMode,
    xManControl  := gvl.gcoils.xWaterValve_HmiOpen,
    xAutoControl := gvl.gcoils.xWaterValve_AutoReq,
    xOutControl  => gvl.gInputs.xWaterValve_Out
);
                
END_PROGRAM

FUNCTION FC_ModbusToRealSwapped : REAL
VAR_INPUT
    wWord1   : WORD;   (* Первое слово из Modbus (например, 53126) *)
    wWord2   : WORD;   (* Второе слово из Modbus (например, 0) *)
END_VAR
VAR
    dwTarget : DWORD;  (* Буфер для сборки 32-битного значения *)
    wTemp1   : WORD;   (* Временные переменные для перестановки байт *)
    wTemp2   : WORD;
    pReal    : POINTER TO REAL; (* Указатель для копирования памяти *)
END_VAR

                  
(* 1. Переставляем байты внутри каждого слова *)
wTemp1 := ROR(wWord1, 8); (* 0xED0C станет 0x0CED *)
wTemp2 := ROR(wWord2, 8); (* 0x0000 останется 0x0000 *)

(* 2. Собираем DWORD в режиме Little-Endian (wTemp2 сдвигаем в старшие биты) *)
dwTarget := SHL(WORD_TO_DWORD(wTemp2), 16) OR WORD_TO_DWORD(wTemp1);
(* На выходе соберется строка 0x41CD0000 *)

(* 3. Копируем область памяти в REAL *)
pReal := ADR(dwTarget);
FC_ModbusToRealSwapped := pReal^;
                
END_FUNCTION

(*
    ФУНКЦИЯ: F_GetReal_BADC
    ОПИСАНИЕ: Разбор REAL 32 бита из 2 регистров WORD, порядок байт BADC.

    Прибор передаёт байты в порядке: B A D C
    (где ABCD = нормальный Big-Endian порядок)

    Раскладка по байтам:
      pSrc[0] = B,  pSrc[1] = A,  pSrc[2] = D,  pSrc[3] = C

    Для Little-Endian ЦПУ нужно собрать DCBA:
      pDst[0] = C = pSrc[3]
      pDst[1] = D = pSrc[2]
      pDst[2] = A = pSrc[1]
      pDst[3] = B = pSrc[0]
*)
FUNCTION F_GetReal_BADC : REAL
VAR_INPUT
    pBuf : POINTER TO ARRAY[0..1] OF WORD;
END_VAR
VAR
    dw   : DWORD;
    pSrc : POINTER TO BYTE;
    pDst : POINTER TO BYTE;
END_VAR

                  
pSrc    := ADR(pBuf^[0]);
pDst    := ADR(dw);
pDst[0] := pSrc[3]; // C
pDst[1] := pSrc[2]; // D
pDst[2] := pSrc[1]; // A
pDst[3] := pSrc[0]; // B
SysMemCpy(pDest := ADR(F_GetReal_BADC), pSrc := ADR(dw), udiCount := 4);
                
END_FUNCTION

PROGRAM InfluxUdpSender
VAR
		fbSender: FB_InfluxUdpSender;
	fbBuf    : FB_InfluxBuffer;
	sendData : STRING(5000); // Data to send
	sIP : STRING :='192.168.150.133'; // InfluxIP
    uiPort : UINT := 8089; // Influx port
	sParam:STRING(200);
END_VAR

                  		sendData := 'CEX15,title=aliy2s_app511_abak_101_172 ';

// Initialization (Measurement mariyu Tag set cheyadam)
// =============================================================
fbBuf(sMeasurement:= 'CEX15', sTagKey:= 'title', sTagValue:= 'aliy2s_app511_abak_101_172');

fbBuf.AddReal('rPosValveDiazo',   GVL.gInputRegs.rPosValveDiazo);
fbBuf.AddReal('rPosValveSoda',   GVL.gInputRegs.rPosValveSoda);
fbBuf.AddReal('rPosValveSteam',   GVL.gInputRegs.rPosValveSteam);

fbBuf.AddReal('rPhApp511',   GVL.gInputRegs.rPhApp511);

fbBuf.AddReal('rTempApp511',   GVL.gInputRegs.rTempApp511);

fbBuf.AddReal('WE_1_app_511',   GVL.gInputRegs.WE_1);

fbBuf.AddReal('WE_2_app_511',   GVL.gInputRegs.WE_2);


fbBuf.AddReal('TotalWater_511',   GVL.gInputRegs.IR_TotalWater);

fbBuf.AddReal('TotalSoda_511',   GVL.gInputRegs.IR_TotalSoda);


fbBuf.AddReal('FlowSoda_511',   GVL.gInputRegs.IR_FlowSoda);

fbBuf.AddReal('FlowWater_511',   GVL.gInputRegs.IR_FlowWater);
// Send Data

// =============================================================
fbSender(sSendData:= fbBuf.sBuffer, sIPInflux:= sIP, uiPortInflux:= uiPort);
                
END_PROGRAM

FUNCTION_BLOCK FB_InfluxBuffer
VAR_INPUT
    sMeasurement : STRING(80);   // Measurement name (e.g., 'CEX6')
    sTagKey      : STRING(40);   // Tag name (e.g., 'title')
    sTagValue    : STRING(80);   // Tag value (e.g., 'kolonna_23b')
END_VAR

VAR_OUTPUT
    sBuffer      : STRING(5000); // Resulting string for fbSender
END_VAR

VAR
    iCurrentLen  : INT;          // Current length of sBuffer
END_VAR

                  // Initialization: Clear buffer and add Measurement + Tag
// Format: "Measurement,TagKey=TagValue " (note the space at the end)
sBuffer := CONCAT(sMeasurement, ',');
sBuffer := CONCAT(sBuffer, sTagKey);
sBuffer := CONCAT(sBuffer, '=');
sBuffer := CONCAT(sBuffer, sTagValue);
sBuffer := CONCAT(sBuffer, ' '); // Line protocol space between tags and fields

iCurrentLen := LEN(sBuffer);
                

METHOD PUBLIC AddReal : BOOL
VAR_INPUT
    sName : STRING(40);
    rVal  : REAL;
END_VAR
VAR
    sFragment : STRING(100);
END_VAR
                        
// Add comma if not the first field
IF iCurrentLen > (LEN(sMeasurement) + LEN(sTagKey) + LEN(sTagValue) + 3) THEN
    sFragment := ',';
ELSE
    sFragment := '';
END_IF

// Format: Key=Value
sFragment := CONCAT(sFragment, sName);
sFragment := CONCAT(sFragment, '=');
sFragment := CONCAT(sFragment, REAL_TO_STRING(rVal));

// Append to buffer using STU for safety or simple CONCAT
STU.StrConcatA(ADR(sFragment), ADR(sBuffer), SIZEOF(sBuffer));
iCurrentLen := LEN(sBuffer);
AddReal := TRUE;
                      
END_METHOD

METHOD PUBLIC AddDWord : BOOL
VAR_INPUT
    sName : STRING(40);
    dwVal : DWORD;
END_VAR
VAR
    sFragment : STRING(100);
    sTemp     : STRING(20);
END_VAR
                        
// Add comma if not the first field
IF iCurrentLen > (LEN(sMeasurement) + LEN(sTagKey) + LEN(sTagValue) + 3) THEN
    sFragment := ',';
ELSE
    sFragment := '';
END_IF

// Format: Key=Value (DWORD преобразуется в UDINT для строки)
sFragment := CONCAT(sFragment, sName);
sFragment := CONCAT(sFragment, '=');

// Convert DWORD to string
sTemp := DWORD_TO_STRING(dwVal);
sFragment := CONCAT(sFragment, sTemp);

// Append to buffer
STU.StrConcatA(ADR(sFragment), ADR(sBuffer), SIZEOF(sBuffer));
iCurrentLen := LEN(sBuffer);
AddDWord := TRUE;
                      
END_METHOD

METHOD Clear : BOOL
VAR_INPUT
END_VAR
                        // Очистка буфера для нового измерения
sBuffer := CONCAT(sMeasurement, ',');
sBuffer := CONCAT(sBuffer, sTagKey);
sBuffer := CONCAT(sBuffer, '=');
sBuffer := CONCAT(sBuffer, sTagValue);
sBuffer := CONCAT(sBuffer, ' ');

iCurrentLen := LEN(sBuffer);
Clear := TRUE;
                      
END_METHOD
END_FUNCTION_BLOCK

FUNCTION_BLOCK FB_InfluxUdpSender
VAR_INPUT
	sSendData : STRING(2000); // Data to send
    sIPInflux : STRING :='192.168.215.5'; // InfluxIP
    uiPortInflux : UINT := 8089; // Influx port
END_VAR
VAR
	eState: 			CLIENT_STATE;								// Шаг состояния клиента
	
	fbUdpPeer: 			NBS.UDP_Peer;								// ФБ создания UDP-пира
	fbUdpSend: 			NBS.UDP_Send;								// ФБ отправки данных
	sendData : STRING(2000); // Data to send
    numberOfBytesToSend : UDINT := 0; // Number of bytes to send
	influxIP: NBS.IP_ADDR;

	fbSendTrig:			R_TRIG;										// Триггер записи
	
	blinker:BLINK;
	TimeCycle: TIME:= T#10S;
	bStart : BOOL := FALSE;
END_VAR

                  	blinker(ENABLE:=bStart,timelow:=TimeCycle, timehigh:=T#1S);
	
CASE eState OF	

	CLIENT_STATE.CREATE:	// создаем UDP-пира на заданном порту
		
		fbUdpPeer
		(
			xEnable		:= TRUE, 
			ipAddr		:= , 
			uiPort		:= ,
			ipMultiCast	:= ,  
		);
	
		IF fbUdpPeer.xActive THEN
			bStart := TRUE;
			eState	:= CLIENT_STATE.WAITING;
			influxIP.sAddr:=sIPInflux;
		ELSIF fbUdpPeer.xError THEN
			; // обработка ошибок
		END_IF

	CLIENT_STATE.WAITING:	// ожидаем команды на запись
	
		fbSendTrig(CLK:=blinker.OUT);
		
		IF fbSendTrig.Q THEN
// Calculate number of bytes to send
			sendData := sSendData;
			numberOfBytesToSend := DINT_TO_UDINT(Stu.StrLenA(ADR(sendData)));			
			
			eState	:= CLIENT_STATE.SEND;
		END_IF
	
	CLIENT_STATE.SEND:		// отправляем запрос серверу
		
			fbUdpSend
			(
				xExecute	:=	TRUE,
				udiTimeOut:= 1000, 
				hPeer		:=	fbUdpPeer.hPeer, 
				ipAddr:=  influxIP, 
				uiPort:= uiPortInflux, 
				szSize:= numberOfBytesToSend, 
				pData:= ADR(sendData), 
			);
			
			IF (fbUdpSend.xDone OR fbUdpSend.xError) THEN
				fbUdpSend(xExecute:=FALSE);
				eState	:= 	CLIENT_STATE.WAITING;
			END_IF
	
END_CASE
                
END_FUNCTION_BLOCK

FUNCTION_BLOCK FB_ValveS_Compact
VAR_INPUT
    xMode        : BOOL; 
    xManControl  : BOOL; 
    xAutoControl : BOOL; 
END_VAR

VAR_OUTPUT
    xOutControl  : BOOL; 
END_VAR

                  // Компактная реализация в одну строку с помощью SEL
xOutControl := SEL(xMode, xManControl, xAutoControl);
                
END_FUNCTION_BLOCK

(* ИСПРАВЛЕНИЕ v4.1.0:
        - Исправлен разбор lrTotalVolume (LREAL / Double 64 бит).
        - Прибор передаёт регистры в порядке Big-Endian (src[0] = MSW, src[3] = LSW).
        - ЦПУ ПЛК — Little-Endian, поэтому выполняется разворот по WORD-словам:
          pW[3] = src[0] (старший), pW[0] = src[3] (младший).
        - Побайтовый подход заменён на пословный (POINTER TO WORD) — корректнее
          и безопаснее, так как каждый WORD внутри уже находится в правильном
          байтовом порядке аппаратуры Little-Endian.
*)
 
FUNCTION_BLOCK fbElemerREM
VAR_INPUT
    pFlowBuffer         : POINTER TO ARRAY[0..1] OF WORD;  (* Канал 0: Мгновенный расход F2, 2 регистра WORD *)
    pVolumeBuffer       : POINTER TO ARRAY[0..3] OF WORD;  (* Канал 1: Накопленный объём F1, 4 регистра WORD *)
    xCommError          : BOOL;                             (* Признак ошибки связи (из статуса Modbus Slave) *)
    xEnableLog          : BOOL := TRUE;                     (* Флаг разрешения детального логирования на HMI *)
END_VAR
VAR_IN_OUT
    xResetTotalizer     : BOOL;  (* Команда сброса сумматора с HMI — автосброс после выполнения *)
END_VAR
VAR_OUTPUT
    xDataValid          : BOOL;         (* Флаг достоверности данных для контуров ТАУ *)
    rInstantFlow        : REAL;         (* Мгновенный расход F2, куб.м/ч *)
    lrTotalVolume       : LREAL;        (* Накопленный общий объём F1, куб.м *)
    sStatus             : STRING(255);  (* Строка текущего шага для оператора панели *)
END_VAR
VAR
    (* Автомат состояний *)
    eState              : E_REM_State;
    eLastState          : E_REM_State;
 
    (* Указатели для разбора REAL (32 бит) *)
    pByteSrc            : POINTER TO BYTE;
    pByteDst            : POINTER TO BYTE;
    dwRealParser        : DWORD;
 
    (* Указатель для разбора LREAL (64 бит) — пословный разворот *)
    pWordDst            : POINTER TO WORD;  (* Указатель на LREAL как массив из 4 WORD *)
 
    (* Системные таймеры *)
    tonStateTimer       : TON;
    udiMinutesInState   : UDINT;
END_VAR
VAR CONSTANT
    DEVICE_DISCONNECTED : REAL := -10000.0;  (* Маркер аварии датчика *)
END_VAR

                  //==============================================================================
// Расчёт времени нахождения в текущем состоянии (в минутах для HMI)
//==============================================================================
tonStateTimer(IN := (eState = eLastState), PT := T#240h);
udiMinutesInState := TIME_TO_UDINT(tonStateTimer.ET) / 60000;
 
//==============================================================================
// 1. ДИАГНОСТИЧЕСКИЙ КОНТРОЛЬ АВАРИЙ СВЯЗИ ВЕРХНЕГО УРОВНЯ
//==============================================================================
IF xCommError THEN
    eState := E_REM_State.ERROR_COMM;
ELSIF xResetTotalizer AND eState <> E_REM_State.ERROR_COMM THEN
    eState := E_REM_State.RESET_LOGIC;
ELSIF eState <> E_REM_State.ERROR_COMM AND eState <> E_REM_State.RESET_LOGIC THEN
    eState := E_REM_State.OPERATING;
END_IF;
 
//==============================================================================
// 2. СТРУКТУРА СТЕЙТ-МАШИНЫ
//==============================================================================
CASE eState OF
 
    E_REM_State.INIT: //--------------------------------------------------------
        sStatus        := 'ЭЛЕМЕР-РЭМ: Ожидание первого скана и данных от Modbus-каналов';
        rInstantFlow   := DEVICE_DISCONNECTED;
        lrTotalVolume  := LREAL#-10000.0;
        xDataValid     := FALSE;
 
        IF pFlowBuffer <> 0 AND pVolumeBuffer <> 0 AND NOT xCommError THEN
            eState := E_REM_State.OPERATING;
        END_IF;
 
 
    E_REM_State.OPERATING: //---------------------------------------------------
        sStatus := 'ЭЛЕМЕР-РЭМ: Данные успешно обновляются, идёт технологический учёт';
 
        IF pFlowBuffer <> 0 AND pVolumeBuffer <> 0 THEN
 
            // ----------------------------------------------------------------
            // РАЗБОР МГНОВЕННОГО РАСХОДА F2
            // Канал 0, REAL 32 бита, формат прибора DCBA (Big-Endian)
            // Побайтовый разворот → Little-Endian ЦПУ ПЛК
            // ----------------------------------------------------------------
            pByteSrc := ADR(pFlowBuffer^[0]);
            pByteDst := ADR(dwRealParser);
 
            IF pByteSrc <> 0 AND pByteDst <> 0 THEN
                pByteDst[0] := pByteSrc[3]; // D → LSB
                pByteDst[1] := pByteSrc[2]; // C
                pByteDst[2] := pByteSrc[1]; // B
                pByteDst[3] := pByteSrc[0]; // A → MSB
                SysMemCpy(pDest := ADR(rInstantFlow), pSrc := ADR(dwRealParser), udiCount := SIZEOF(rInstantFlow));
            END_IF;
 
 
            // ----------------------------------------------------------------
            // РАЗБОР НАКОПЛЕННОГО ОБЪЁМА F1
            // Канал 1, Double/LREAL 64 бита, Big-Endian порядок WORD-регистров:
            //   src[0] = MSW (старший), src[3] = LSW (младший)
            //
            // Алгоритм прибора (из документации):
            //   v  = (uint64_t)src[0] << 48
            //   v |= (uint64_t)src[1] << 32
            //   v |= (uint64_t)src[2] << 16
            //   v |= (uint64_t)src[3]
            //
            // На Little-Endian ЦПУ ПЛК LREAL в памяти хранится так:
            //   pW[0] = LSW (биты  0..15)
            //   pW[1]        (биты 16..31)
            //   pW[2]        (биты 32..47)
            //   pW[3] = MSW (биты 48..63)
            //
            // Поэтому разворачиваем порядок WORD-ов:
            //   pW[3] := src[0]   (MSW прибора → старший WORD LREAL)
            //   pW[2] := src[1]
            //   pW[1] := src[2]
            //   pW[0] := src[3]   (LSW прибора → младший WORD LREAL)
            //
            // Байты ВНУТРИ каждого WORD НЕ трогаем — аппаратура ПЛК
            // уже прочитала их корректно в Little-Endian.
            // ----------------------------------------------------------------
            pWordDst := ADR(lrTotalVolume);
 
            IF pWordDst <> 0 THEN
                pWordDst[3] := pVolumeBuffer^[0]; // MSW прибора → старший WORD
                pWordDst[2] := pVolumeBuffer^[1];
                pWordDst[1] := pVolumeBuffer^[2];
                pWordDst[0] := pVolumeBuffer^[3]; // LSW прибора → младший WORD
            END_IF;
 
 
            // ----------------------------------------------------------------
            // ЗАЩИТА ТАУ: Валидация на NaN
            // ----------------------------------------------------------------
            IF rInstantFlow <> rInstantFlow OR lrTotalVolume <> lrTotalVolume THEN
                sStatus    := 'ЭЛЕМЕР-РЭМ: Критическая ошибка! Считано неопределённое значение NaN.';
                xDataValid := FALSE;
            ELSE
                xDataValid := TRUE;
            END_IF;
 
        ELSE
            sStatus    := 'ЭЛЕМЕР-РЭМ: Внимание, обнаружен нулевой указатель буферов опроса!';
            xDataValid := FALSE;
        END_IF;
 
 
    E_REM_State.RESET_LOGIC: //-------------------------------------------------
        sStatus    := 'ЭЛЕМЕР-РЭМ: Выполняется процедура сброса сумматора по команде оператора';
        xDataValid := TRUE;
 
        IF NOT xResetTotalizer THEN
            eState := E_REM_State.OPERATING;
        END_IF;
 
 
    E_REM_State.ERROR_COMM: //--------------------------------------------------
        sStatus       := 'АВАРИЯ связи: Прибор не отвечает. Проверьте кабель RS-485!';
        rInstantFlow  := DEVICE_DISCONNECTED;
        lrTotalVolume := LREAL#-10000.0;
        xDataValid    := FALSE;
 
        IF NOT xCommError THEN
            eState := E_REM_State.INIT;
        END_IF;
 
END_CASE;
 
 
//==============================================================================
// 3. ДИАГНОСТИЧЕСКОЕ ЛОГИРОВАНИЕ ДЛЯ ОПЕРАТОРА ПАНЕЛИ
//==============================================================================
IF xEnableLog AND (eState <> eLastState) THEN
    eLastState := eState;
    sStatus    := CONCAT(sStatus, CONCAT(' | Прошло времени: ', UDINT_TO_STRING(udiMinutesInState)));
    sStatus    := CONCAT(sStatus, ' мин.');
END_IF;
                
END_FUNCTION_BLOCK

(*  Накопленный объём F1: 4 регистра WORD, Big-Endian Double → REAL  *)
FUNCTION F_ElemerREM_Volume : REAL
VAR_INPUT
    pBuf : POINTER TO ARRAY[0..3] OF WORD;
END_VAR
VAR
    lr   : LREAL;
    pW   : POINTER TO WORD;
END_VAR

                  pW    := ADR(lr);
pW[3] := pBuf^[0];
pW[2] := pBuf^[1];
pW[1] := pBuf^[2];
pW[0] := pBuf^[3];
F_ElemerREM_Volume := LREAL_TO_REAL(lr);
                
END_FUNCTION

(* Мгновенный расход F2: 2 регистра WORD, Big-Endian REAL *)
FUNCTION F_ElemerREM_Flow : REAL
VAR_INPUT
    pBuf : POINTER TO ARRAY[0..1] OF WORD;
END_VAR
VAR
    dw : DWORD;
	END_VAR

                  IF pBuf <> 0 THEN
    // Склеиваем два WORD в один DWORD (старшее слово сдвигаем на 16 бит влево)
    dw := SHL(WORD_TO_DWORD(pBuf^[0]), 16) OR WORD_TO_DWORD(pBuf^[1]);

    // Копируем память "бит-в-бит" из DWORD в REAL
    SysMemCpy(pDest := ADR(F_ElemerREM_Flow), pSrc := ADR(dw), udiCount := 4);
END_IF
                
END_FUNCTION

(*
    ФУНКЦИОНАЛЬНЫЙ БЛОК: FB_WaterLoading
    ВЕРСИЯ: 2.0.0
    ОПИСАНИЕ: Автоматическая загрузка воды заданной дозой.
 
    ЛОГИКА:
      - xStart OFF→ON  : старт → открываем клапан (xAutoControl:=TRUE), фиксируем объём
      - xStart ON→OFF  : прерывание оператором → закрываем клапан (xAutoControl:=FALSE)
      - Доза выполнена : rLoaded >= rDose - rDeadband → закрываем клапан, xStart:=FALSE
 
    ВАЖНО: xMode и xAutoControl — VAR_IN_OUT (прямая ссылка на внешние переменные).
           Присвоение только по триггеру (фронт старта, фронт стопа, завершение дозы).
           В рабочем цикле (xRunning=TRUE) — только обновление rLoaded, клапан не трогаем.
 
    СТАТУСЫ (rStatus):
      0.0 = IDLE
      1.0 = RUNNING
      2.0 = DONE
      3.0 = ABORTED
*)
 (*
    ФУНКЦИОНАЛЬНЫЙ БЛОК: FB_WaterLoading
    ВЕРСИЯ: 2.1.0 (Исправленная)
*)

FUNCTION_BLOCK FB_WaterLoading
VAR_INPUT
    rTotalVolume    : REAL;   (* Текущий объём сумматора расходомера, куб.м *)
    rDose           : REAL;   (* Заданная доза, куб.м *)
    rDeadband       : REAL;   (* Мёртвый остаток для предиктивного закрытия, куб.м *)
END_VAR
VAR_IN_OUT
    xStart          : BOOL;   (* Команда: ON=старт, OFF=стоп/прерывание *)
    xMode           : BOOL;   (* Режим клапана: FALSE=ручной, TRUE=авто *)
    xAutoControl    : BOOL;   (* Автозадание клапана *)
END_VAR
VAR_OUTPUT
    rLoaded         : REAL;   (* Загружено в текущем цикле, куб.м *)
    rStatus         : REAL;   (* 0=IDLE 1=RUNNING 2=DONE 3=ABORTED *)
END_VAR
VAR
    rStartVolume    : REAL;
    xLastStart      : BOOL;
    xRunning        : BOOL;
END_VAR

                  // ----------------------------------------------------------------
// ФРОНТ OFF→ON : СТАРТ ДОЗИРОВАНИЯ
// ----------------------------------------------------------------
IF xStart AND NOT xLastStart THEN
    rStartVolume := rTotalVolume;
    rLoaded      := 0.0;
    xRunning     := TRUE;
    rStatus      := 1.0;
    xMode        := TRUE;   // переключаем клапан в авторежим
    xAutoControl := TRUE;   // открываем клапан
END_IF;

// ----------------------------------------------------------------
// РАБОЧИЙ ЦИКЛ: Считаем объем и проверяем достижение дозы
// ----------------------------------------------------------------
IF xRunning THEN
    rLoaded := rTotalVolume - rStartVolume;

    // Доза выполнена — предиктивное закрытие (Высший приоритет)
    IF rLoaded >= (rDose - rDeadband) THEN
        xAutoControl := FALSE;  // закрываем клапан
        xRunning     := FALSE;
        xStart       := FALSE;  // автосброс команды
        rStatus      := 2.0;    // DONE
    END_IF;
END_IF;

// ----------------------------------------------------------------
// ФРОНТ ON→OFF : ПРЕРЫВАНИЕ ОПЕРАТОРОМ
// (Сработает только если доза ЕЩЕ НЕ выполнена в этом цикле)
// ----------------------------------------------------------------
IF NOT xStart AND xLastStart AND xRunning THEN
    xRunning     := FALSE;
    xAutoControl := FALSE;  // закрываем клапан
    rStatus      := 3.0;    // ABORTED
END_IF;

// ----------------------------------------------------------------
// БУФЕР ФРОНТА (в конце скана)
// ----------------------------------------------------------------
xLastStart := xStart;
                
END_FUNCTION_BLOCK

FUNCTION_BLOCK FB_UniversalSteamValveControl
VAR_INPUT
    xEnable       : BOOL;   // Переключатель контура (ВКЛ/ВЫКЛ) [1]
    rTempActual   : REAL;   // Текущая температура [1]
    rSetpoint     : REAL;   // Уставка температуры [1]
    xReset        : BOOL;   // Сброс ошибки ПИД [1]
    
    // Настройки ПИД (передаются снаружи для универсальности)
    rKp           : REAL;   
    rTn           : REAL;   
    rTv           : REAL;   
    rLimitLow     : REAL;   
    rLimitHigh    : REAL;   
END_VAR

VAR_IN_OUT
    // Переменные IN_OUT изменяют внешнюю переменную по ссылке
    rValveOut     : REAL;   // Управляющее воздействие на клапан (0-100% или иное) [3]
    xAutoModeCmd  : BOOL;   // Команда режима: TRUE = АВТО, FALSE = РУЧНОЙ
END_VAR

VAR_OUTPUT
    xStatusActive : BOOL;   // Статус работы контура [1]
END_VAR

VAR
    fbPID         : oscat_basic.CTRL_PID; // Экземпляр ПИД из библиотеки Oscat [1]
    xOldEnable    : BOOL;   // Для детектора фронта [1]
    rInternalY    : REAL;   // Промежуточная переменная для выхода PID
END_VAR

                  
// --- ЛОГИКА ---

// 1. Управление режимами (детектирование изменения xEnable)
IF xEnable AND NOT xOldEnable THEN
    // ВКЛЮЧЕНИЕ:
    xStatusActive := TRUE;       // [2]
    xAutoModeCmd  := TRUE;       // Переводим внешний флаг в режим АВТО
    
ELSIF NOT xEnable AND xOldEnable THEN
    // ВЫКЛЮЧЕНИЕ:
    xStatusActive := FALSE;      // [2]
    xAutoModeCmd  := FALSE;      // Снимаем флаг АВТО (переход в ручной)
    rValveOut     := 0.0;        // Обнуляем выход на клапан [2]
END_IF;

xOldEnable := xEnable;

// 2. Вызов ПИД-регулятора
fbPID(
    ACT := rTempActual,          // [2]
    SET := rSetpoint,            // [2]
    MAN := NOT xStatusActive,    // Если не активен, ПИД в ручном режиме (MAN=TRUE) [2]
    RST := xReset,               // [2]
    KP  := rKp,                  // [2]
    TN  := MAX(rTn, 1.0),        // Защита от деления на 0, как в источнике [2]
    TV  := rTv,                  // [3]
    LL  := rLimitLow,            // [3]
    LH  := rLimitHigh            // [3]
);

// 3. Передача значения из ПИД во внешнюю переменную через IN_OUT
// Обновляем выход только если контур активен, чтобы не перебивать ручное управление при выключенном блоке
IF xStatusActive THEN
    rValveOut := fbPID.Y;        // [3]
END_IF;
                
END_FUNCTION_BLOCK

PROGRAM PRG_Apparatus511
VAR
    // Экземпляр функционального блока управления клапаном пара
    fbSteamControl_511 : FB_UniversalSteamValveControl;

    // Переменные для связи с HMI (если они еще не заданы в GVL)
    xEnableTempControl : BOOL;  // Команда с HMI: Включить автоматическое поддержание температуры
    rTempSetpoint_511  : REAL;  // Задание поддерживаемой температуры в аппарате (до 100 °C)
    xResetTempPID      : BOOL;  // Команда сброса ошибки ПИД-регулятора

    // Промежуточная переменная для связи флагов режима
    xSteamAutoMode     : BOOL;  // TRUE = АВТО, FALSE = РУЧНОЙ
END_VAR

                  // --- ВЫЗОВ БЛОКА ПОДДЕРЖАНИЯ ТЕМПЕРАТУРЫ АППАРАТА 511 ---

fbSteamControl_511(
    xEnable       := xEnableTempControl,          // Команда оператора на запуск контура
    rTempActual   := GVL.gInputRegs.rTempApp511,  // Текущая температура из аппарата 511 [3, 4]
    rSetpoint     := rTempSetpoint_511,           // Уставка температуры (до 100 °C) [5, 6]
    xReset        := xResetTempPID,               // Сброс ПИД
    
    // IN_OUT переменные (передаются по ссылке напрямую)
    rValveOut     := GVL.gHoldingRegs.rAutoSet_Steam, // Запись выхода ПИД в авто-задание клапана пара [1, 2]
    xAutoModeCmd  := xSteamAutoMode                   // Получаем команду режима от ФБ
);

// --- СИНХРОНИЗАЦИЯ РЕЖИМОВ УПРАВЛЕНИЯ ---
// Согласно вашей логике, клапан пара (fbValveSteam) работает в ручном режиме 
// когда GVL.gCoils.xManualMode_Steam = TRUE [2].
// Поскольку наш ФБ выдает TRUE для режима АВТО, нам нужно инвертировать этот сигнал:
GVL.gCoils.xManualMode_Steam := NOT xSteamAutoMode;
                
END_PROGRAM

(*Рабочий алгоритм этого блока будет следующим: по переднему фронту сигнала xStart он включает внутренний пид-регулятор, который открывает клапан и начинает нагрев. Если xKeepTemp = FALSE, то как только текущая температура достигает заданной, мы снимаем сигнал разрешения (xEnable) и внутреннего пид-регулятора (нагрев прекращается). Если xKeepTemp = TRUE, то регулятор продолжает поддерживать температуру, пока активен xStart.
*)
FUNCTION_BLOCK FB_AutoHeater
VAR_INPUT
    xStart        : BOOL;   // Признак запуска нагрева (по переднему фронту)
    xKeepTemp     : BOOL;   // TRUE = поддерживать температуру после достижения, FALSE = отключить после нагрева (разовая операция)
    rTempActual   : REAL;   // Текущая температура в аппарате
    rTargetTemp   : REAL;   // Целевая температура, до которой нужно нагреть (или уставка)
    rTolerance    : REAL := 0.5; // Зона чувствительности (нагрев считается завершенным при Т >= уставка - Tolerance)
    // Параметры пид-регулятора
    rKp           : REAL := 1.0;
    rTn           : REAL := 10.0;
    rTv           : REAL := 0.0;
END_VAR
VAR_IN_OUT
    rValveOut     : REAL;   // Управляющее воздействие на клапан (0..100%)
    xAutoModeCmd  : BOOL;   // Выбор режима (TRUE = авто, FALSE = ручной)
END_VAR
VAR_OUTPUT
    xActive       : BOOL;   // Состояние: нагрев в процессе
    xDone         : BOOL;   // Состояние: нагрев успешно завершен (целевая Т достигнута)
END_VAR
VAR
    fbSteamControl : FB_UniversalSteamValveControl;
    xOldStart      : BOOL;  // Память сигнала запуска
    xEnablePID     : BOOL;  // Внутренний сигнал работы пид-регулятора
END_VAR

                  // --- 1. Обработка команд и переходов состояний ---
// Детектор переднего фронта запуска: если пришел сигнал Start
IF xStart AND NOT xOldStart THEN
    xActive    := TRUE;   // Начинаем нагрев
    xDone      := FALSE;  // Сбрасываем флаг готовности
    xEnablePID := TRUE;   // Разрешаем работу внутреннего регулятора
END_IF;

// Условие достижения температуры
IF xActive AND (rTempActual >= (rTargetTemp - rTolerance)) THEN
    xDone := TRUE;   // Сигнализируем успешное достижение уставки
    
    // Если НЕ нужно удерживать температуру, выключаем нагрев
    IF NOT xKeepTemp THEN
        xActive    := FALSE;  // Останавливаем процесс
        xEnablePID := FALSE;  // Отключаем ПИД-регулятор
    END_IF;
END_IF;

// Обработка ручного сброса / выключения
IF NOT xStart THEN
    xDone := FALSE; // Сбрасываем статус при снятии Start
    IF xActive THEN
        xActive    := FALSE;
        xEnablePID := FALSE;
    END_IF;
END_IF;

xOldStart := xStart; // Запоминаем состояние фронта

// --- 2. Вызов регулирующего функционального блока ---
fbSteamControl(
    xEnable       := xEnablePID,
    rTempActual   := rTempActual,
    rSetpoint     := rTargetTemp,
    xReset        := FALSE,
    rValveOut     := rValveOut,
    xAutoModeCmd  := xAutoModeCmd
);
                
END_FUNCTION_BLOCK

PROGRAM PRG_Apparatus511_Heating
VAR
    // Экземпляр нашего блока автоматического нагрева
    fbAutoHeater511 : FB_AutoHeater;

    // Вспомогательная переменная для связи флагов режима клапана
    xSteamAutoMode  : BOOL; 
END_VAR

                  // --- Автоматический нагрев аппарата 511 ---
fbAutoHeater511(
// --- Входы управления с HMI ---
xStart        := GVL.gCoils.xStartHeating_511,      // Признак запуска нагрева с панели оператора
xKeepTemp     := GVL.gCoils.xKeepTempHeating_511,   // TRUE = поддерживать температуру после достижения
rTargetTemp   := GVL.gHoldingRegs.rSetTempApp511,   // Уставка целевой температуры (до 100 °C)
// --- Технологические параметры ---
rTempActual   := GVL.gInputRegs.rTempApp511,        // Фактическая температура в емкости
rTolerance    := 0.5,                               // Допуск в градусах
// --- Настройки пид ---
rKp           := GVL.gHoldingRegs.rKp_Steam_511,
rTn           := GVL.gHoldingRegs.rTn_Steam_511,
rTv           := GVL.gHoldingRegs.rTv_Steam_511,
// --- Выходы на исполнительные механизмы (IN_OUT) ---
rValveOut     := GVL.gHoldingRegs.rAutoSet_Steam,   
xAutoModeCmd  := xSteamAutoMode
);
                
END_PROGRAM

FUNCTION_BLOCK FB_AutoCouplingDrainCascade
VAR_INPUT
    xStart             : BOOL;   // Триггер запуска стадии
    
    // --- Параметры Диазосоединения ---
    rFlowDiazoActual   : REAL;   // Текущий мгновенный расход диазо (м3/ч)
    rFlowDiazoSetpoint : REAL;   // Заданный мгновенный расход диазо
    
    // --- Параметры pH ---
    rPhActual          : REAL;   // Текущий pH (9.5..12 ед.)
    rPhSetpoint        : REAL;   // Уставка поддерживаемого pH
    
    // --- Условия завершения (Опустошение) ---
    rZeroFlowThreshold : REAL := 0.2;   // Порог "отсутствия расхода" (< 0.2 м3/ч)
    tEmptyDelay        : TIME := T#20S; // Время подтверждения отсутствия расхода
    
    // --- Настройки ПИД ---
    rKp_Diazo          : REAL := 1.0;
    rTn_Diazo          : REAL := 5.0;
    rTv_Diazo          : REAL := 0.0;
    rKp_pH             : REAL := 2.0;
    rTn_pH             : REAL := 10.0;
    rTv_pH             : REAL := 0.0;
END_VAR

VAR_IN_OUT
    rValveOutDiazo     : REAL;   // Задание на клапан диазо (0..100%)
    xAutoModeCmdDiazo  : BOOL;   // Режим АВТО для диазо
    rValveOutSoda      : REAL;   // Задание на клапан соды (0..100%)
    xAutoModeCmdSoda   : BOOL;   // Режим АВТО для соды
END_VAR

VAR_OUTPUT
    xActive            : BOOL;   // Стадия идет
    xDone              : BOOL;   // Стадия успешно завершена
    
    // --- Переменные для HMI ---
    rTimeLeft          : REAL;   // Оставшееся время до завершения (сек)
    rStateCode         : REAL;   // Код текущего состояния (0.0 .. 4.0)
    sStateStr          : STRING; // Текстовая расшифровка состояния
END_VAR

VAR
    fbPidFlowDiazo     : oscat_basic.CTRL_PID;
    fbPidPh            : oscat_basic.CTRL_PID;
    tonEmptyTimer      : TON;
    
    iState             : INT := 0; // Внутренний регистр шага State Machine
    xOldStart          : BOOL;
    xNeedStop          : BOOL;   // Флаг однократного останова оборудования
END_VAR

                  
// --- ЛОГИКА БЛОКА ---

// 1. Детектор старта (Исправление №1: Явный сброс выходов при старте)
IF xStart AND NOT xOldStart THEN
    iState     := 1;    // Переход в RUNNING
    xActive    := TRUE; // Явное включение
    xDone      := FALSE;// Явный сброс готовности
    xNeedStop  := FALSE;// Явный сброс команды останова
    
    xAutoModeCmdDiazo := TRUE;
    xAutoModeCmdSoda  := TRUE;
END_IF;

// 2. Детектор прерывания оператором
IF NOT xStart AND xOldStart AND (iState = 1 OR iState = 2) THEN
    iState := 4; // Переход в ABORTED
    xNeedStop := TRUE;
END_IF;

// 3. Вызов таймера опустошения
// Таймер работает ТОЛЬКО когда мы находимся на шаге 2 (EMPTYING)
tonEmptyTimer(
    IN := (iState = 2), 
    PT := tEmptyDelay
);

// 4. КОНЕЧНЫЙ АВТОМАТ (STATE MACHINE)
CASE iState OF
    0: // --- IDLE (Ожидание) ---
        sStateStr  := 'ОЖИДАНИЕ: Аппарат готов к запуску';
        rStateCode := 0.0;
        xActive    := FALSE;
        xDone      := FALSE;
        rTimeLeft  := TIME_TO_REAL(tEmptyDelay) / 1000.0; 

    1: // --- RUNNING (Нормальное регулирование) ---
        sStateStr  := 'РАБОТА: Поддержание расхода и pH';
        rStateCode := 1.0;
        xActive    := TRUE;
        xDone      := FALSE;
        rTimeLeft  := TIME_TO_REAL(tEmptyDelay) / 1000.0;
        
        // Условие перехода: расход упал ниже порога
        IF rFlowDiazoActual <= rZeroFlowThreshold THEN
            iState := 2; 
        END_IF;

    2: // --- EMPTYING (Фиксация отсутствия расхода) ---
        sStateStr  := 'ВНИМАНИЕ: Падение расхода, отсчет времени...';
        rStateCode := 2.0;
        xActive    := TRUE;
        
        // Исправление №2: Безопасное вычитание времени (защита от переполнения/отрицательного результата)
        IF tonEmptyTimer.ET < tEmptyDelay THEN
            rTimeLeft := TIME_TO_REAL(tEmptyDelay - tonEmptyTimer.ET) / 1000.0;
        ELSE
            rTimeLeft := 0.0;
        END_IF;
        
        // Возврат в работу: если расход "ожил" (насос снова захватил жидкость)
        IF rFlowDiazoActual > rZeroFlowThreshold THEN
            iState := 1; 
            
        // Успешное завершение: таймер досчитал до конца
        ELSIF tonEmptyTimer.Q THEN
            iState := 3;
            xNeedStop := TRUE; // Даем команду на закрытие клапанов
        END_IF;

    3: // --- DONE (Успешное завершение) ---
        sStateStr  := 'ЗАВЕРШЕНО: Емкость диазосоединения пуста';
        rStateCode := 3.0;
        xActive    := FALSE;
        xDone      := TRUE;
        rTimeLeft  := 0.0;
        
        // Исправление №3: Защита от гонки состояний при быстром повторном старте
        IF NOT xStart AND NOT xOldStart THEN
            iState := 0;
        END_IF;

    4: // --- ABORTED (Прервано оператором) ---
        sStateStr  := 'ПРЕРВАНО: Остановка по команде оператора';
        rStateCode := 4.0;
        xActive    := FALSE;
        xDone      := FALSE;
        rTimeLeft  := 0.0;
        
        // Исправление №3: Защита от гонки состояний при быстром повторном старте
        IF NOT xStart AND NOT xOldStart THEN
            iState := 0;
        END_IF;

END_CASE;

// 5. Вызов ПИД-регуляторов (Работают только на активных шагах 1 и 2)
IF iState = 1 OR iState = 2 THEN
    fbPidFlowDiazo(
        ACT := rFlowDiazoActual, SET := rFlowDiazoSetpoint,
        MAN := FALSE, RST := FALSE, KP := rKp_Diazo, TN := MAX(rTn_Diazo, 1.0),
        TV := rTv_Diazo, LL := 0.0, LH := 100.0
    );
    rValveOutDiazo := fbPidFlowDiazo.Y;

    fbPidPh(
        ACT := rPhActual, SET := rPhSetpoint,
        MAN := FALSE, RST := FALSE, KP := rKp_pH, TN := MAX(rTn_pH, 1.0),
        TV := rTv_pH, LL := 0.0, LH := 100.0
    );
    rValveOutSoda := fbPidPh.Y;
END_IF;

// 6. Однократный безопасный останов
IF xNeedStop THEN
    // Сбрасываем интеграторы ПИД
    fbPidFlowDiazo(MAN := TRUE, SET := 0.0, ACT := 0.0, RST := TRUE);
    fbPidPh(MAN := TRUE, SET := 0.0, ACT := 0.0, RST := TRUE);
    
    // Закрываем клапаны и возвращаем в ручной режим
    rValveOutDiazo    := 0.0;
    xAutoModeCmdDiazo := FALSE;
    rValveOutSoda     := 0.0;
    xAutoModeCmdSoda  := FALSE;
    
    xNeedStop := FALSE; // Сбрасываем триггер останова
END_IF;

xOldStart := xStart;
                
END_FUNCTION_BLOCK

PROGRAM PRG_Apparatus511_CascadeDrain
VAR
    // Экземпляр последней версии блока (с конечным автоматом)
    fbCascadeDrain511 : FB_AutoCouplingDrainCascade;
    
    // Вспомогательные переменные для инверсии ручного/автоматического режимов
    xDiazoAutoMode    : BOOL;
    xSodaAutoMode     : BOOL;
END_VAR

                  
// --- 1. ВЫЗОВ АЛГОРИТМА СЛИВА С ПОДДЕРЖАНИЕМ pH ---
fbCascadeDrain511(
    // Управление
    xStart             := GVL.gCoils.xStartCoupling_511,       
    
    // Параметры Диазосоединения
    rFlowDiazoActual   := GVL.gInputRegs.IR_FlowDiazo,         // Мгновенный расход [1]
    rFlowDiazoSetpoint := GVL.gHoldingRegs.rSetFlowDiazo_511,  // Уставка расхода [1]
    
    // Параметры pH
    rPhActual          := GVL.gInputRegs.rPhApp511,            // Показания pH-метра [1]
    rPhSetpoint        := GVL.gHoldingRegs.rSetPh_511,         // Целевая уставка pH [1]
    
    // Настройки условия завершения (конвертация UINT секунд в TIME)
    rZeroFlowThreshold := GVL.gHoldingRegs.rZeroFlowThreshold_511, 
    tEmptyDelay        := UDINT_TO_TIME(UINT_TO_UDINT(GVL.gHoldingRegs.uiEmptyDelaySec_511) * 1000), 
    
    // Прямая связь с авто-заданиями физических клапанов (IN_OUT)
    rValveOutDiazo     := GVL.gHoldingRegs.rAutoSet_Diazo,     // [3]
    xAutoModeCmdDiazo  := xDiazoAutoMode,
    
    rValveOutSoda      := GVL.gHoldingRegs.rAutoSet_Soda,      // [3]
    xAutoModeCmdSoda   := xSodaAutoMode
);

// --- 2. СИНХРОНИЗАЦИЯ РЕЖИМОВ (Ручной/Авто) ---
// В физической логике клапанов TRUE = Ручной режим, поэтому инвертируем команду от блока
GVL.gCoils.xManualMode_Diazo := NOT xDiazoAutoMode;
GVL.gCoils.xManualMode_Soda  := NOT xSodaAutoMode;

// --- 3. ПЕРЕДАЧА СТАТУСОВ КОНЕЧНОГО АВТОМАТА НА HMI ---
// Булевые лампочки состояния процесса
GVL.gCoils.xCouplingActive_511 := fbCascadeDrain511.xActive; 
GVL.gCoils.xCouplingDone_511   := fbCascadeDrain511.xDone;   

// Числовые коды, оставшееся время и текст
GVL.gInputRegs.rTimeLeft_511   := fbCascadeDrain511.rTimeLeft;  // Оставшиеся секунды при падении расхода
GVL.gInputRegs.rStateCode_511  := fbCascadeDrain511.rStateCode; // 0.0, 1.0, 2.0, 3.0, 4.0
GVL.sStateStr_511              := fbCascadeDrain511.sStateStr;  // Расшифровка этапа
                
END_PROGRAM

CONFIGURATION Application
  RESOURCE Application ON PLC
(* global variable list GVL *)
{attribute 'qualified_only'}


VAR_GLOBAL
	
	gInputRegs	:	InputRegs;
	gHoldingRegs	:	HoldingRegs;
	gInputs	:	Inputs;
	gCoils	:	Coils;
    // =========================================================================
    // АНАЛОГОВЫЕ ВХОДЫ (Опрос датчиков)
    // =========================================================================
    rPressPump207v      : REAL; // Давление насоса мембранного 207в (0.5..6 кгс/см2)
    rTempApp511         : REAL; // Температура реакционной среды в аппарате 511 (до 100 °C)
    rPhApp511           : REAL; // Показания pH-метра аппарата 511 (9.5..12 ед.)

	
	WE_1_s:WORD;
	WE_1_f:WORD;
	
	WE_2_s:WORD;
	WE_2_f:WORD;
	
	sStateStr_511:string(255);
	
	
	
	
	
	
	
	
	
	
	
	
	
	
	
	
	
	
	
	
	
	
	
    // =========================================================================
    // СЧЕТЧИКИ И РАСХОДОМЕРЫ (Опрос текущего расхода и накопленного объема)
    // =========================================================================
    rFlowDiazo          : REAL; // Текущий расход диазосоединения (м3/ч)
    rTotalDiazo         : REAL; // Накопленный объем диазосоединения (м3)
    
    rFlowSoda           : REAL; // Текущий расход едкого натра 14% (м3/ч)
    rTotalSoda          : REAL; // Накопленный объем едкого натра 14% (м3)
    
    rFlowWater          : REAL; // Текущий расход воды артезианской/деминерализованной (м3/ч)
    rTotalWater         : REAL; // Накопленный объем воды / счетчик дозы (м3)

    // =========================================================================
    // СИГНАЛЫ СОСТОЯНИЯ КЛАПАНОВ (Входы обратной связи)
    // =========================================================================
    rPosValveDiazo      : REAL; // Сигнализация положения (% открытия) клапана диазосоединения
    rPosValveSoda       : REAL; // Сигнализация положения (% открытия) клапана едкого натра
    rPosValveSteam      : REAL; // Сигнализация положения (% открытия) клапана пара
    
    xStsValveWaterOpen  : BOOL; // Сигнализатор положения отсечного пневмокрана воды - ОТКРЫТ
    xStsValveWaterClose : BOOL; // Сигнализатор положения отсечного пневмокрана воды - ЗАКРЫТ

    // =========================================================================
    // АНАЛОГОВЫЕ И ДИСКРЕТНЫЕ ВЫХОДЫ (Управление исполнительными механизмами)
    // =========================================================================
    rCmdValveDiazo  AT  %QW0    : WORD; // Управление регулирующим клапаном диазосоединения (0..100%)
    rCmdValveSoda   AT  %QW1    : WORD; // Управление регулирующим клапаном едкого натра (0..100%)
    rCmdValveSteam  AT  %QW2    : WORD; // Управление регулирующим клапаном пара для поддержания температуры (0..100%)
    xCmdValveWater      : BOOL; // Дискретное управление отсечным пневмокраном воды (закрытие при достижении дозы)

    // =========================================================================
    // ПЕРЕМЕННЫЕ HMI / СЕНСОРНОЙ ПАНЕЛИ (Уставки и задания)
    // =========================================================================
    rSpTempApp511       : REAL; // Задание поддерживаемой температуры в аппарате (до 100 °C)
    rSpFlowDiazo        : REAL; // Задание необходимого расхода диазосоединения (до 19 м3/ч)
    rSpFlowSoda         : REAL; // Задание необходимого расхода едкого натра (до 7.35 м3/ч)
    rSpDoseWater        : REAL; // Задание необходимой дозы воды (до 7.35 м3/ч)
    
    // Переменные для алгоритма дозирования щелочи
    rSpPhLow            : REAL := 9.2; // Нижний порог pH для увеличения открытия клапана щелочи
    rSpPhHigh           : REAL := 9.7; // Верхний порог pH для уменьшения открытия клапана щелочи
    rSpPhTargetMatch    : REAL := 9.6; // Порог pH для открытия клапана щелочи на стадии "сочетания"
    rSpPhTargetClose    : REAL := 9.5; // Порог pH для закрытия клапана щелочи
MDS_3RTD_1_start_ad : POINTER TO ARRAY[0..10] OF WORD;;
END_VAR
(* global variable list PVL *)
{attribute 'qualified_only'}
VAR_GLOBAL PERSISTENT RETAIN
	rHoldingRegs: HoldingRegs;
END_VAR
    TASK MainTask(INTERVAL := T#20ms, PRIORITY := 1);
    TASK InfluxTask(INTERVAL := T#20ms, PRIORITY := 1);
    TASK HmiCommunication(INTERVAL := T#100ms, PRIORITY := 21);
    TASK Task_Bus(INTERVAL := T#20ms, PRIORITY := 1);
    TASK Task_can(INTERVAL := T#20ms, PRIORITY := 1);
    PROGRAM PLC_PRG WITH MainTask : PLC_PRG;
    PROGRAM ASK_prg WITH MainTask : ASK_prg;
    PROGRAM PRG_Valves WITH MainTask : PRG_Valves;
    PROGRAM PRG_Apparatus511_Heating WITH MainTask : PRG_Apparatus511_Heating;
    PROGRAM InfluxUdpSender WITH InfluxTask : InfluxUdpSender;
    PROGRAM PLC_PRG_MBS_TCP_SLAVE WITH HmiCommunication : PLC_PRG_MBS_TCP_SLAVE;
  END_RESOURCE
END_CONFIGURATION
